FUNCTION "FC_IoMapOutputs" : Void
{ S7_Optimized_Access := 'TRUE' }
VERSION : 0.1

// Pick & Place — Copyright (C) 2026 Jeferson Tramonti
// Licenciado sob a GNU GPLv3 — veja o arquivo LICENSE.

// Mapeamento de SAIDAS fisicas (%Q/%QD) a partir de duas fontes.
// FC stateless, chamada no FIM do scan pelo OB_Main. Isola TODO o enderecamento
// fisico de saida num ponto unico (principio §6 da arquitetura) e aplica a
// mascara de estado seguro nas saidas de processo.
//
// ULTIMA barreira fisica de safety:
//  - Em i_SafeState: M1/M2 := 0.0, Grab/RotCW/RotCCW := FALSE (garantido mesmo
//    que um FB a montante falhe em se auto-proteger).
//  - GripCW/GripCCW := FALSE SEMPRE (gripper nao usado).
//  - Luzes NAO mascaradas (precisam indicar emergencia/parado).
//  - SP de eixo NAO mascarado (FB_AxisPos ja congela; forcar 0 V seria movimento perigoso).

    VAR_INPUT
        i_SafeState : Bool;   // FB_MachineMode.o_SafeState (E-Stop OU Stop OU Falha)
        i_Red : Bool;   // -> %Q0.4
        i_Green : Bool;   // -> %Q0.5
        i_Yellow : Bool;   // -> %Q0.6
        i_ResetLite : Bool;   // -> %Q0.3
        i_StartLite : Bool;   // -> %Q0.7
        i_StopLite : Bool;   // -> %Q1.0
        i_RotCW : Bool;   // FB_PickPlaceSeq.o_RotCW  -> %Q1.2
        i_RotCCW : Bool;   // FB_PickPlaceSeq.o_RotCCW -> %Q1.4
    END_VAR

    VAR_IN_OUT
        io_Station : "typeStation";   // le Sts.M1Speed/M2Speed/VacuumOn/AxisX.SP/AxisZ.SP
    END_VAR

    VAR_OUTPUT
        o_ResetLite : Bool;   // %Q0.3
        o_Red : Bool;   // %Q0.4
        o_Green : Bool;   // %Q0.5
        o_Yellow : Bool;   // %Q0.6
        o_StartLite : Bool;   // %Q0.7
        o_StopLite : Bool;   // %Q1.0
        o_Grab : Bool;   // %Q1.1
        o_RotCW : Bool;   // %Q1.2
        o_GripCW : Bool;   // %Q1.3 (sempre FALSE)
        o_RotCCW : Bool;   // %Q1.4
        o_GripCCW : Bool;   // %Q1.5 (sempre FALSE)
        o_M1 : Real;   // %QD30 — saida analogica (Real)
        o_M2 : Real;   // %QD34 — saida analogica (Real)
        o_Xsp : Real;   // %QD38 — saida analogica (Real)
        o_Zsp : Real;   // %QD42 — saida analogica (Real)
    END_VAR

    VAR_TEMP
        t_bothRot : Bool;     // conflito RotCW & RotCCW
    END_VAR

BEGIN

    REGION Sinalizacao
    // Luzes: repasse direto do VAR_INPUT, SEM mascara (devem indicar emergencia/parado)
        #o_ResetLite := #i_ResetLite;
        #o_Red := #i_Red;
        #o_Green := #i_Green;
        #o_Yellow := #i_Yellow;
        #o_StartLite := #i_StartLite;
        #o_StopLite := #i_StopLite;
    END_REGION

    REGION Processo
    // M1/M2/Grab: mascara de estado seguro (zera/desliga em emergencia)
        IF #i_SafeState THEN
            #o_M1 := 0.0;
            #o_M2 := 0.0;
            #o_Grab := FALSE;
        ELSE
        // LReal (DB) -> Real (%QD): estreitamento explicito (valores 0-10 V cabem em Real)
            #o_M1 := LREAL_TO_REAL(#io_Station.Sts.M1Speed);
            #o_M2 := LREAL_TO_REAL(#io_Station.Sts.M2Speed);
            #o_Grab := #io_Station.Sts.VacuumOn;
        END_IF;
    END_REGION

    REGION Rotacao
    // Mascara + exclusao mutua (conflito -> estado seguro: ambos FALSE)
        #t_bothRot := #i_RotCW AND #i_RotCCW;
        IF #i_SafeState OR #t_bothRot THEN
            #o_RotCW := FALSE;
            #o_RotCCW := FALSE;
        ELSE
            #o_RotCW := #i_RotCW;
            #o_RotCCW := #i_RotCCW;
        END_IF;
    END_REGION

    REGION Setpoints
    // SP de eixo: SEM mascara (FB_AxisPos ja congela; FC so repassa)
    // LReal (DB) -> Real (%QD): estreitamento explicito
        #o_Xsp := LREAL_TO_REAL(#io_Station.Sts.AxisX.SP);
        #o_Zsp := LREAL_TO_REAL(#io_Station.Sts.AxisZ.SP);
    END_REGION

    REGION GripperOff
    // Gripper nao usado no projeto — intertravamento sempre FALSE
        #o_GripCW := FALSE;
        #o_GripCCW := FALSE;
    END_REGION

END_FUNCTION

